TYPE ST_P1MesData :
STRUCT
	sDMC_Code			:STRING;
	nOP_Index			:INT;
	sOP_Name			:STRING;
	sOP_CustomData		:STRING(1000);
	sOP_ReceipeList		:STRING(1000);
END_STRUCT
END_TYPE

(* stored: Version 1.1.0.1, ProductVersion 3.1.4024.10
   DUT ST_P1MesData: Id {8196b4d2-c69f-474d-82e6-32ff3660ea41} *)
